PROGRAM Camera
VAR
		cameraData : CameraConnectionUDP;
END_VAR

cameraData();

END_PROGRAM

(* stored: Version 1.1.0.1, ProductVersion 3.1.4024.11
   POU Camera: Id {e90280ff-791e-436e-94db-5e32a5133a14}, SpecialFunc None *)
